Yaskawa INFORM job: TEST1.JBI

/JOB
//NAME TEST1
//POS
///NPOS 1,0,0,1,0,0
///TOOL 0
///POSTYPE PULSE
///PULSE
C00000=390876,202089,35618,0,-117424,182917
///POSTYPE BASE
///RECTAN
///RCONF 0,0,0,0,0,0,0,0,0,0,0,0,0,0,0,0,0,0,0,0,0,0,0,0
P00100=0.000,0.000,0.000,0.0000,0.0000,0.0000
//ARGINFO
///ARGTYPE B,B,B,I,I,,,
///COMMENT
Arg1
Arg2
Arg3
Arg4
Arg5
Arg6
Arg7
Arg8
//INST
///DATE 2020/11/19 13:27
///ATTR SC,RW
///GROUP1 RB1
///LVARS 0,0,0,0,0,5,0,0
NOP
'COMMENT
SET LP000 P100
IMOV LP000 V=201.0
IFTHENEXP B003=0
	'No Wait
ELSEIFEXP B003=1
	'Wait for Signal
	 WAIT IN#(B004)=ON
ELSE
	'Wait for Timer
	 TIMER T=LI005
ENDIF
END
